// TIA Portal V19 export
DATA_BLOCK "Block_2_DB"   // DB2
// stored: InstanceOfName Block_2, InstanceOfType FB
"Block_2"
   // VAR
   //    HF : Array[0..10] of Bool;
   // END_VAR
BEGIN
END_DATA_BLOCK
